Fanuc KAREL source: kb00172.KL

PROGRAM KB00172
%NOLOCKGROUP
%ENVIRONMENT IOSETUP
VAR
P1:INTEGER;P2:INTEGER;P3 : STRING[80];P4:INTEGER
BEGIN
--
--
--
P1=1
P2=1
P3='A'
P4=1
SET_PORT_CMT(P1,P2,P3,P4)
END KB00172
